Omron CX-Programmer project NewProject (CX-Programmer 9.51)

# PLC my_first_project: CP1L L
; Comment

## Program NewProgram1 (cyclic task 0)
Local symbols
Start W0.01 BOOL
button_1 0.00 BOOL  ; Comment
button_2 0.01 BOOL  ; Comment
out_2 100.01 BOOL  ; Comment
out_3 100.02 BOOL  ; Comment

### Section Section1

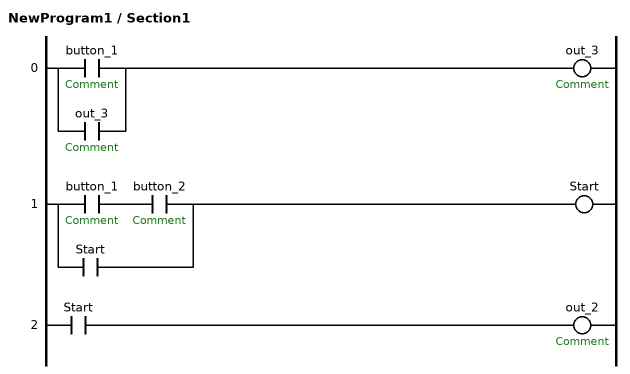
; rung 0
LD button_1  ; Comment
OR out_3  ; Comment
OUT out_3  ; Comment
; rung 1
LD button_1  ; Comment
AND button_2  ; Comment
OR Start
OUT Start
; rung 2
LD Start
OUT out_2  ; Comment

### Section END
; rung 0
END(001)